# EPICS StreamDevice protocol: siteApps/cryomodule-1-0/proto/oda.proto
# Toyotech Power Supply Unipolar Communication Protocol
# Data format
# 	baud rate: 9600
#	start: 1
#	data: 8
#	stop: 1
#	parity: None
#	hardware handshake: None
# Communication Procedure
# Transmit: Mnemonics[and parameters] <CR>[<LF>]
# Receive: <ACK><CR><LF>
# Transmit: <ENQ>
# Receive: Measurement values or parameters <CR>

Terminator = LF;

#InTerminator  = LF;
#OutTerminator = LF;
ReplyTimeout = 3000;

#-----------------------------------------------#
setRemote
{
	out "SYST:REM";
}

setLocal
{
	out "SYST:LOC";
}

setChannel
{
	out "INST %s";
}
setChannelRB
{
	out "INST?"; in "%s";
}

setOutput
{
	out "OUTP %s";
}
setOutputRB
{
	out "OUTP?"; in "%b";
}

#-----------------------------------------------#
setVoltage
{
	out "VOLT %g";
}

setVoltageRB
{
	out "VOLT?"; in "%f";
}

getVoltage
{
	out "MEAS:VOLT?"; in "%f";
}

#-----------------------------------------------#
setCurrent
{
	out "CURR %g";
}

setCurrentRB
{
	out "CURR?"; in "%f";
}

getCurrent
{
	out "MEAS:CURR?"; in "%f";
}
#-----------------------------------------------#
